(*
A list implementation for managing `I_Arg`.  
*)
INTERFACE I_ArgList EXTENDS I_Debug

(*
Provides the maximum capacity of the list.
*)
PROPERTY Cap : UDINT
GET
END_GET
END_PROPERTY

(*
Retrieves the `I_Arg` at the specified index.  
Returns:
- `Ok` - Successfully retrieves the `I_Arg`.
- `Err.Idx` - The specified index is out of bounds.
- `Err.InvRef` - Invalid output reference.
- `Err.Idx` - `iOut` = 0.
*)
METHOD Get : Result
VAR_INPUT
	nIndex		: UDINT;
	iOut		: REFERENCE TO I_Arg;
END_VAR
END_METHOD

END_INTERFACE

(* stored: Version 1.1.0.1
   Itf I_ArgList: Id {ebf0d78f-4078-4420-90cf-3c27fe88901b}
   Property Cap: Id {93fc02a4-69a8-48a7-b684-8b0e8d2a39cd}
   Get Get: Id {20d25a38-c36a-42c3-bd92-88fa4e743bf1}
   Method Get: Id {f2f87690-f9cb-4ae6-a2f0-8e33ef6f803d} *)
